FUNCTION_BLOCK PUBLIC FB_LampOnOff IMPLEMENTS I_Subject
VAR
	nLightLevel			:	USINT;
	_ipObserver			:	I_Observer;	
END_VAR

METHOD Attach
VAR_INPUT
	ipObserver		: I_Observer;
END_VAR
IF (ipObserver = 0) THEN
	RETURN;
END_IF
_ipObserver := ipObserver;
END_METHOD

METHOD Detach
_ipObserver := 0;
END_METHOD

// Sets the control value to 0.
METHOD PUBLIC Off
nLightLevel := 0;
IF (_ipObserver <> 0) THEN
	_ipObserver.Update(nLightLevel);
END_IF
END_METHOD

// Sets the control value to 100.
METHOD PUBLIC On
nLightLevel := 100;
IF (_ipObserver <> 0) THEN
	_ipObserver.Update(nLightLevel);
END_IF
END_METHOD

END_FUNCTION_BLOCK

(* stored: Version 1.1.0.1, ProductVersion 3.1.4024.12
   POU FB_LampOnOff: Id {55e66dc1-05c3-43f8-9bc8-5075ca0cd865}, SpecialFunc None
   Method Attach: Id {37e3754b-e80b-4217-ae1f-9f5d2206bf53}
   Method Detach: Id {aadac412-1d51-49a6-96cd-c8bde1a89977}
   Method Off: Id {54f23483-66d0-4707-9581-54558ff84187}
   Method On: Id {ea9cd1d9-8590-4b0b-b6ec-c19fb0ca1b1d} *)
